{attribute 'linkalways'} 
{attribute 'no_explicit_call' := 'This FB is a CLASS and must be accessed using methods or properties'}
{attribute 'enable_dynamic_creation'}
FUNCTION_BLOCK Node_F_VN_FillContainerExp_SINT EXTENDS VisionNode
VAR
    ipContainer : _ITcVnContainer;
    nValue : _SINT(0);
    nStartIdx : _ULINT(0);
    nCount : _ULINT(0);
    hrPrev : _HRESULT(S_OK);
    hresult : _HRESULT(S_OK);
END_VAR

METHOD PUBLIC  Clone : I_Node
VAR
    pNode : POINTER TO Node_F_VN_FillContainerExp_SINT;
END_VAR
pNode := __NEW(Node_F_VN_FillContainerExp_SINT);
Clone := pNode^;
END_METHOD

METHOD FB_init : BOOL
VAR_INPUT
    bInitRetains : BOOL; // if TRUE, the retain variables are initialized (warm start / cold start)
    bInCopyCode : BOOL;  // if TRUE, the instance afterwards gets moved into the copy code (online change)
END_VAR
AddInput('ipContainer', ipContainer);
AddInput('nValue', nValue);
AddInput('nStartIdx', nStartIdx);
AddInput('nCount', nCount);
AddInput('hrPrev', hrPrev);
AddOutput('ipContainer', ipContainer);
AddOutput('hresult',hresult);
END_METHOD

METHOD PROTECTED OnExecute : HRESULT
hresult.Value := F_VN_FillContainerExp_SINT(
    ipContainer := ipContainer.Value,
    nValue := nValue.Value,
    nStartIdx := nStartIdx.Value,
    nCount := nCount.Value,
    hrPrev:= hrPrev.Value);
END_METHOD

METHOD PUBLIC PreExecutionCheck
VAR_INPUT
    Check : I_PreExecutionChecks;
END_VAR
Check.IsTrue(ipContainer.IsValid, 'ipContainer must be a valid container');
Check.IsTrue(ipContainer.HasType(TC_GLOBAL_CONST_LIST.ContainerType_Vector_SINT), 'ipContainer contains incorrect type');
END_METHOD

END_FUNCTION_BLOCK

(* stored: Version 1.1.0.1, ProductVersion 3.1.4024.13
   POU Node_F_VN_FillContainerExp_SINT: Id {ec23ee48-9959-47ef-9572-cb0317c05df7}, SpecialFunc None
   Folder Constructor: Id {d2acf7fb-fca3-4c8c-8e6c-cfcf7bcd0224}
   Method Clone: Id {d1d4bf44-6e2e-4fff-8a87-d5a6a0339581}
   Method FB_init: Id {199a0d43-f4e4-4720-982f-2785db636071}
   Method OnExecute: Id {0a6b3efd-383d-4481-92d4-5f628b1badb3}
   Method PreExecutionCheck: Id {e0a9933e-1ad2-482a-aeca-03fb15a27fb6} *)
